(*
SPDX-FileCopyrightText: © 2026 Oleksandr Tiutyk <trofimich@gmail.com>
SPDX-License-Identifier: MIT
License: https://opensource.org/license/mit
*)

{attribute 'enable_dynamic_creation'}	
{attribute 'no_explicit_call' := 'do not call this function block directly'} 
FUNCTION_BLOCK EmptyException EXTENDS Exception IMPLEMENTS IEmptyException
VAR
	{attribute 'hide'} 
	_ClassName : STRING := __POUNAME();
END_VAR

{attribute 'monitoring' := 'call'}
PROPERTY ClassName : REFERENCE TO STRING
GET
ClassName REF= _ClassName;
END_GET
END_PROPERTY

METHOD Clone : IObject
VAR
	exceptionClone : POINTER TO EmptyException;
END_VAR
exceptionClone := __NEW(EmptyException);

IF exceptionClone = 0 THEN
	DynamicMemoryManager.RaiseAllocationFailure();
	RETURN;
END_IF

Clone := exceptionClone^;
END_METHOD

{attribute 'monitoring' := 'call'}
PROPERTY Empty : BOOL
GET
Empty := TRUE;
END_GET
END_PROPERTY

METHOD GetMessage : ERROR_MESSAGE
VAR_INPUT
	showSource : BOOL := FALSE;
	timestampDisplayMode : TIMESTAMP_DISPLAY_MODE := TIMESTAMP_DISPLAY_MODE.HIDDEN;
END_VAR
GetMessage := "";
END_METHOD

METHOD FINAL GetRootException : IException
GetRootException := THIS^;
END_METHOD

{attribute 'monitoring' := 'call'}
PROPERTY NamespaceName : REFERENCE TO STRING
GET
NamespaceName REF= CurrentNamespace.Name;
END_GET
END_PROPERTY

{attribute 'monitoring' := 'call'}
PROPERTY SelfSize : ULINT
GET
SelfSize := XSIZEOF(THIS^);
END_GET
END_PROPERTY

{attribute 'monitoring' := 'call'}
PROPERTY FINAL Severity : ERROR_SEVERITY
GET
Severity := ERROR_SEVERITY.ERROR;
END_GET
END_PROPERTY

METHOD FINAL ToError
VAR_IN_OUT CONSTANT
	targetError : ERROR;
END_VAR
VAR_INPUT
	severity : ERROR_SEVERITY;	
END_VAR
VAR
	i : DINT;
	
	innerException : IException;
END_VAR
IF NOT __ISVALIDREF(targetError) THEN
	RETURN;
END_IF

targetError.Clear();
END_METHOD

END_FUNCTION_BLOCK

(* stored: Version 1.1.0.1
   POU EmptyException: Id {244a2959-0232-440a-847e-a759a1a08774}, SpecialFunc None
   Property ClassName: Id {f1e26cf2-22eb-4c46-8fbb-0a6918bd4e41}
   Get Get: Id {0717f242-d57a-488d-bd81-79b911bf33a8}
   Method Clone: Id {bdb7f31b-80ac-4a36-949e-72042507cf19}
   Property Empty: Id {3a478482-003d-459c-be74-6269eef6c595}
   Get Get: Id {3dc40e6e-e146-41bb-95ff-60840a3e2a14}
   Method GetMessage: Id {d392dbf0-15ed-4bc4-b890-d88d59c980b5}
   Method GetRootException: Id {b66f953d-5d5f-4b95-8b56-529c01f62adf}
   Property NamespaceName: Id {ee6c054c-3239-4728-9ab1-ac21e0fcddd1}
   Get Get: Id {0d4169e1-e8c7-494b-8c7d-c0efd72d4924}
   Property SelfSize: Id {3756ad03-0622-4800-b508-023f372e0d54}
   Get Get: Id {ffbcebbf-243e-4d68-ada3-a836de091da7}
   Property Severity: Id {353b0aa3-e49b-4f0e-b0ec-42e56a9bd9bb}
   Get Get: Id {63789ae6-08e5-4bee-820b-b4785cbb43fb}
   Method ToError: Id {ec0a50b6-9055-426a-a59c-7629d8b077e3} *)
